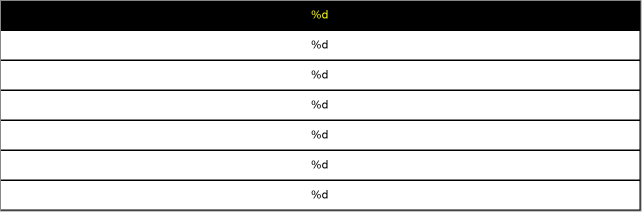
VISUALIZATION CARTON_FORMING_SHIFT_ELEMENT  // 642x212
VAR_INPUT
	index:		UDINT;
END_VAR
    Rectangle (0,0 640x30), "%d", text variable: wu_cartonForming_shiftRegister_debug.shift_debug[index].step_id
    Rectangle (0,30 640x30), "%d", text variable: wu_cartonForming_shiftRegister_debug.shift_debug[index].status.0, colour toggle: wu_cartonForming_shiftRegister_debug.shift_debug[index].status.0
    Rectangle (0,90 640x30), "%d", text variable: wu_cartonForming_shiftRegister_debug.shift_debug[index].reject_reason
    Rectangle (0,120 640x30), "%d", text variable: wu_cartonForming_shiftRegister_debug.shift_debug[index].status.4, colour toggle: wu_cartonForming_shiftRegister_debug.shift_debug[index].status.4
    Rectangle (0,180 640x30), "%d", text variable: wu_cartonForming_shiftRegister_debug.shift_debug[index].equipment_number
    Rectangle (0,150 640x30), "%d", text variable: wu_cartonForming_shiftRegister_debug.shift_debug[index].status.5, colour toggle: wu_cartonForming_shiftRegister_debug.shift_debug[index].status.5
    Rectangle (0,60 640x30), "%d", text variable: wu_cartonForming_shiftRegister_debug.shift_debug[index].status.1, colour toggle: wu_cartonForming_shiftRegister_debug.shift_debug[index].status.1
END_VISUALIZATION

(* stored: Version 1.1.0.1, ProductVersion 3.1.4024.3
   Visu CARTON_FORMING_SHIFT_ELEMENT: Id {ccbd81c9-ee8c-4f11-a05a-47cac6bde6ff} *)
